// SIMATIC STEP 7 (V5.x) project T13 E 30
// CPU: CPU313 C-2 DP(1)
// station: P_ADR_BUS
// station: Hardware
// station: Equipo SIMATIC 300
// program: Programa S7(1)

SYMBOL_TABLE
"AUXILIARES"	DB 1	DB 1
"MARCHA"	I 0.0	BOOL
"F. CARRERA"	I 0.1	BOOL
"CELULA"	I 0.2	BOOL
"PARO"	I 0.3	BOOL
"Cycle Execution"	OB 1	OB 1
"CINTA TRANS."	Q 0.0	BOOL
"LED CINTA"	Q 0.1	BOOL
"MOTOR TALADRO"	Q 0.2	BOOL
"PISTON EXPANDIDO"	Q 0.3	BOOL
"LED PISTON EXP."	Q 0.4	BOOL
"LED PARO"	Q 0.5	BOOL
END_SYMBOL_TABLE

DATA_BLOCK "AUXILIARES"	// DB 1
VERSION : 0.1
  STRUCT
   F0 : BOOL ;
   F1 : BOOL ;
   F2 : BOOL ;
   F3 : BOOL ;
   F4 : BOOL ;
   F5 : BOOL ;
   F6 : BOOL ;
   F7 : BOOL ;
   B10 : BOOL ;
   B11 : BOOL ;
   B12 : BOOL ;
   B13 : BOOL ;
  END_STRUCT ;	
BEGIN
END_DATA_BLOCK

ORGANIZATION_BLOCK "Cycle Execution"	// OB 1
TITLE = "Main Program Sweep (Cycle)"
//TALADRADORA AUTOMATIZADA.
VERSION : 0.1
VAR_TEMP
  OB1_EV_CLASS : BYTE ;	//Bits 0-3 = 1 (Coming event), Bits 4-7 = 1 (Event class 1)
  OB1_SCAN_1 : BYTE ;	//1 (Cold restart scan 1 of OB 1), 3 (Scan 2-n of OB 1)
  OB1_PRIORITY : BYTE ;	//Priority of OB Execution
  OB1_OB_NUMBR : BYTE ;	//1 (Organization block 1, OB1)
  OB1_RESERVED_1 : BYTE ;	//Reserved for system
  OB1_RESERVED_2 : BYTE ;	//Reserved for system
  OB1_PREV_CYCLE : INT ;	//Cycle time of previous OB1 scan (milliseconds)
  OB1_MIN_CYCLE : INT ;	//Minimum cycle time of OB1 (milliseconds)
  OB1_MAX_CYCLE : INT ;	//Maximum cycle time of OB1 (milliseconds)
  OB1_DATE_TIME : DATE_AND_TIME ;	//Date and time OB1 started
END_VAR
BEGIN
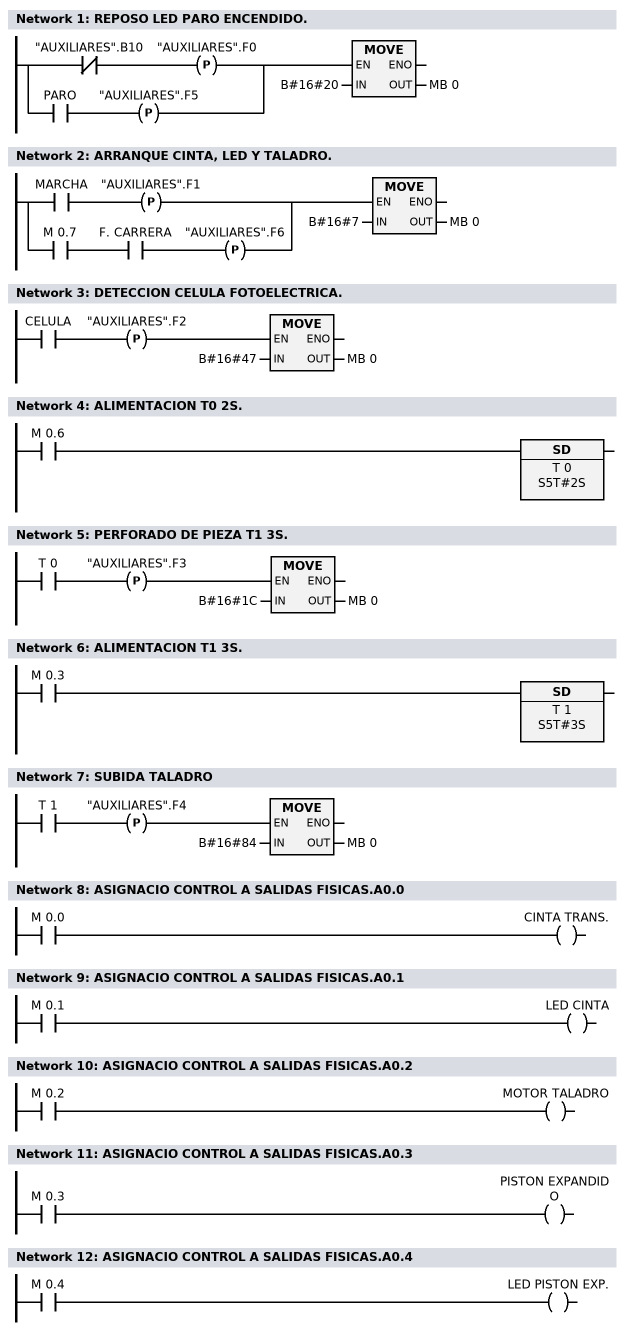
NETWORK
TITLE = REPOSO LED PARO ENCENDIDO.
      A(;
      AN    "AUXILIARES".B10;
      FP    "AUXILIARES".F0;
      O(;
      A     "PARO";
      FP    "AUXILIARES".F5;
      );
      );
      JNB   _001;
      L     B#16#20;
      T     MB 0;
_001: NOP   0;
NETWORK
TITLE = ARRANQUE CINTA, LED Y TALADRO.
      A(;
      A     "MARCHA";
      FP    "AUXILIARES".F1;
      O(;
      A     M 0.7;
      A     "F. CARRERA";
      FP    "AUXILIARES".F6;
      );
      );
      JNB   _002;
      L     B#16#7;
      T     MB 0;
_002: NOP   0;
NETWORK
TITLE = DETECCION CELULA FOTOELECTRICA.
//UTILIZO M0.6 PARA ALIMENTAR T0.
      A     "CELULA";
      FP    "AUXILIARES".F2;
      JNB   _003;
      L     B#16#47;
      T     MB 0;
_003: NOP   0;
NETWORK
TITLE = ALIMENTACION T0 2S.
      A     M 0.6;
      L     S5T#2S;
      SD    T 0;
NETWORK
TITLE = PERFORADO DE PIEZA T1 3S.
      A     T 0;
      FP    "AUXILIARES".F3;
      JNB   _004;
      L     B#16#1C;
      T     MB 0;
_004: NOP   0;
NETWORK
TITLE = ALIMENTACION T1 3S.
      A     M 0.3;
      L     S5T#3S;
      SD    T 1;
NETWORK
TITLE = SUBIDA TALADRO
//ACTIVO M0.7 PARA QUE GOBIERNE F.CARRERA TA QUE ESTARA PRESIONADO EN REPOSO.
      A     T 1;
      FP    "AUXILIARES".F4;
      JNB   _005;
      L     B#16#84;
      T     MB 0;
_005: NOP   0;
NETWORK
TITLE = ASIGNACIO CONTROL A SALIDAS FISICAS.A0.0
      A     M 0.0;
      =     "CINTA TRANS.";
NETWORK
TITLE = ASIGNACIO CONTROL A SALIDAS FISICAS.A0.1
      A     M 0.1;
      =     "LED CINTA";
NETWORK
TITLE = ASIGNACIO CONTROL A SALIDAS FISICAS.A0.2
      A     M 0.2;
      =     "MOTOR TALADRO";
NETWORK
TITLE = ASIGNACIO CONTROL A SALIDAS FISICAS.A0.3
      A     M 0.3;
      =     "PISTON EXPANDIDO";
NETWORK
TITLE = ASIGNACIO CONTROL A SALIDAS FISICAS.A0.4
      A     M 0.4;
      =     "LED PISTON EXP.";
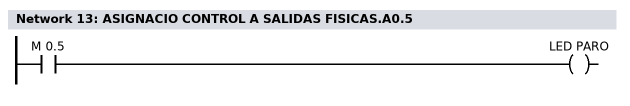
NETWORK
TITLE = ASIGNACIO CONTROL A SALIDAS FISICAS.A0.5
      A     M 0.5;
      =     "LED PARO";
END_ORGANIZATION_BLOCK
